FUNCTION_BLOCK FB_MqttCom_String
VAR_INPUT
	(* published message *)
	sTopicPub : STRING(255) := 'MyTopic_String';
	sPayloadPub : STRING(255);
	sTopicSub : STRING(255) := 'MyTopic_String';
END_VAR

VAR_OUTPUT
	{attribute 'TcEncoding':='UTF-8'}
	sPayloadRcv : STRING(255);
END_VAR

VAR
	fbMqttClient : FB_IotMqttClient;
	bSetParameter : BOOL := TRUE;
	bConnect : BOOL := TRUE;
	
	
	i: UDINT;
	fbTimer : TON := (PT:=T#1S);
	
	(* received message *)
	bSubscribed : BOOL;
	{attribute 'TcEncoding':='UTF-8'}
	sTopicRcv : STRING(255);

	fbMessageQueue : FB_IotMqttMessageQueue;
	fbMessage : FB_IotMqttMessage;
	
	hrErrorOccurred : HRESULT; // contains the latest occurred error
END_VAR

IF bSetParameter THEN
	bSetParameter := FALSE;
	fbMqttClient.sHostName:= 'localhost';
	fbMqttClient.nHostPort:= 1883;
//	fbMqttClient.sClientId:= 'MyTcMqttClient'; 
	fbMqttClient.sTopicPrefix:= ''; 
	fbMqttClient.ipMessageQueue := fbMessageQueue;
END_IF

fbMqttClient.Execute(bConnect);
IF fbMqttClient.bError THEN
	// add your error logging here
	hrErrorOccurred := fbMqttClient.hrErrorCode;
END_IF

IF fbMessageQueue.nQueuedMessages > 0 THEN
	IF fbMessageQueue.Dequeue(fbMessage:=fbMessage) THEN
		fbMessage.GetTopic(pTopic:=ADR(sTopicRcv), nTopicSize:=SIZEOF(sTopicRcv) );
		fbMessage.GetPayload(pPayload:=ADR(sPayloadRcv), nPayloadSize:=SIZEOF(sPayloadRcv), bSetNullTermination:=FALSE);
	END_IF
END_IF

IF fbMqttClient.bConnected THEN
	IF NOT bSubscribed THEN
		bSubscribed := fbMqttClient.Subscribe(sTopic:=sTopicSub, eQoS:=TcIotMqttQos.AtMostOnceDelivery);
		IF fbMqttClient.bError THEN
			// add your error logging here
			hrErrorOccurred := fbMqttClient.hrErrorCode;
		END_IF
	END_IF
	fbTimer(IN:=TRUE);
	IF fbTimer.Q THEN // publish new payload every second
		fbTimer(IN:=FALSE);
		fbMqttClient.Publish(	sTopic:= sTopicPub, 
								pPayload:= ADR(sPayloadPub), nPayloadSize:= LEN2(ADR(sPayloadPub))+1, 
								eQoS:= TcIotMqttQos.AtMostOnceDelivery, bRetain:= FALSE, bQueue:= FALSE );
		IF fbMqttClient.bError THEN
			// add your error logging here
			hrErrorOccurred := fbMqttClient.hrErrorCode;
		END_IF
	END_IF
END_IF

END_FUNCTION_BLOCK

(* stored: Version 1.1.0.1, ProductVersion 3.1.4024.11
   POU FB_MqttCom_String: Id {0d8ba684-9101-4eaf-bbb6-cd32c51e551b}, SpecialFunc None *)
